{attribute addProperty BoxType "EK1100-0000-0018"}
{attribute addProperty Id "Beckhoff_ELXxxxxEK1122Beckhoff_ELXxxxxEK1122_CE175A58162A_0001_ELX1052_0000_0016ELX1052_0A1DBF07648A_0002_ELX1054_0000_0016ELX1054_FE7182BE12816A_0003_ELX1058_0000_0016ELX1058_F462A61522428A_0004_ELX2002_0000_0016ELX2002_B180A8D3405A_0005_ELX2008_0000_0016ELX2008_04E0E56B8811A_0006_ELX3152_0000_0016ELX3152_1C870F0C16020A_0007_ELX3152_0000_0017ELX3152_1C870F0C16020A_0008_ELX3152_0090_0016ELX3152_1C870F0C16020A_0009_ELX3152_0090_0017ELX3152_1C870F0C16020A_0010_ELX3158_0000_0016ELX3158_91E9C02235244A_0011_ELX3181_0000_0016ELX3181_02AD9A7917622A_0012_ELX3181_0000_0017ELX3181_02AD9A7917622A_0013_ELX3202_0000_0016ELX3202_0EB9D2E916020A_0014_ELX3202_0090_0016ELX3202_0EB9D2E916020A_0015_ELX3204_0000_0016ELX3204_5DC9EB4C22428A_0016_ELX3204_0090_0016ELX3204_5DC9EB4C22428A_0017_ELX3252_0000_0016ELX3252_F145ADB416020A_0018_ELX3312_0000_0016ELX3312_5B7A95F016020A_0019_ELX3312_0090_0016ELX3312_5B7A95F016020A_0020_ELX3314_0000_0016ELX3314_2E54E3B022428A_0021_ELX3314_0090_0016ELX3314_2E54E3B022428A_0022_ELX3351_0000_0016ELX3351_537A111616020A_0023_ELX3351_0090_0016ELX3351_537A111616020A_0024_ELX4154_0000_0016ELX4154_253CF8AE15219A_0025_ELX4181_0000_0016ELX4181_E6374D8B15219A_0026_ELX4181_0000_0017ELX4181_E6374D8B15219A_0027_ELX5151_0000_0016ELX5151_347031A716020A_0028_ELX5151_0090_0016ELX5151_347031A716020A_0030_ELX9410_0000_0016ELX9410_D787878A486A_0031_ELX9410_0000_0017ELX9410_D787878A486A_0032_ELX9410_0000_0018ELX9410_AF51CCF7486A_0033_ELX9560_0000_0016ELX9560_FB68D8D1486A_0034_ELX9560_0000_0017ELX9560_FB68D8D1486A_0035_ELX9560_0000_0018ELX9560_E7D0746E486"}
{attribute addProperty CRC "818935286"}
{attribute addProperty SizeInBites "4984"}
{attribute addProperty SizeInBytes "623"}
TYPE Beckhoff_ELXxxxx_30CFF5F6 EXTENDS EK1100_179A0949 :
STRUCT
	{attribute addProperty Name "Beckhoff_ELXxxxxEK1122"}
	Beckhoff_ELXxxxxEK1122 : Beckhoff_ELXxxxxEK1122_CE175A58;
	{attribute addProperty Name "A_0001_ELX1052_0000_0016"}
	A_0001_ELX1052_0000_0016 : ELX1052_0A1DBF07;
	{attribute addProperty Name "A_0002_ELX1054_0000_0016"}
	A_0002_ELX1054_0000_0016 : ELX1054_FE7182BE;
	{attribute addProperty Name "A_0003_ELX1058_0000_0016"}
	A_0003_ELX1058_0000_0016 : ELX1058_F462A615;
	{attribute addProperty Name "A_0004_ELX2002_0000_0016"}
	A_0004_ELX2002_0000_0016 : ELX2002_B180A8D3;
	{attribute addProperty Name "A_0005_ELX2008_0000_0016"}
	A_0005_ELX2008_0000_0016 : ELX2008_04E0E56B;
	{attribute addProperty Name "A_0006_ELX3152_0000_0016"}
	A_0006_ELX3152_0000_0016 : ELX3152_1C870F0C;
	{attribute addProperty Name "A_0007_ELX3152_0000_0017"}
	A_0007_ELX3152_0000_0017 : ELX3152_1C870F0C;
	{attribute addProperty Name "A_0008_ELX3152_0090_0016"}
	A_0008_ELX3152_0090_0016 : ELX3152_1C870F0C;
	{attribute addProperty Name "A_0009_ELX3152_0090_0017"}
	A_0009_ELX3152_0090_0017 : ELX3152_1C870F0C;
	{attribute addProperty Name "A_0010_ELX3158_0000_0016"}
	A_0010_ELX3158_0000_0016 : ELX3158_91E9C022;
	{attribute addProperty Name "A_0011_ELX3181_0000_0016"}
	A_0011_ELX3181_0000_0016 : ELX3181_02AD9A79;
	{attribute addProperty Name "A_0012_ELX3181_0000_0017"}
	A_0012_ELX3181_0000_0017 : ELX3181_02AD9A79;
	{attribute addProperty Name "A_0013_ELX3202_0000_0016"}
	A_0013_ELX3202_0000_0016 : ELX3202_0EB9D2E9;
	{attribute addProperty Name "A_0014_ELX3202_0090_0016"}
	A_0014_ELX3202_0090_0016 : ELX3202_0EB9D2E9;
	{attribute addProperty Name "A_0015_ELX3204_0000_0016"}
	A_0015_ELX3204_0000_0016 : ELX3204_5DC9EB4C;
	{attribute addProperty Name "A_0016_ELX3204_0090_0016"}
	A_0016_ELX3204_0090_0016 : ELX3204_5DC9EB4C;
	{attribute addProperty Name "A_0017_ELX3252_0000_0016"}
	A_0017_ELX3252_0000_0016 : ELX3252_F145ADB4;
	{attribute addProperty Name "A_0018_ELX3312_0000_0016"}
	A_0018_ELX3312_0000_0016 : ELX3312_5B7A95F0;
	{attribute addProperty Name "A_0019_ELX3312_0090_0016"}
	A_0019_ELX3312_0090_0016 : ELX3312_5B7A95F0;
	{attribute addProperty Name "A_0020_ELX3314_0000_0016"}
	A_0020_ELX3314_0000_0016 : ELX3314_2E54E3B0;
	{attribute addProperty Name "A_0021_ELX3314_0090_0016"}
	A_0021_ELX3314_0090_0016 : ELX3314_2E54E3B0;
	{attribute addProperty Name "A_0022_ELX3351_0000_0016"}
	A_0022_ELX3351_0000_0016 : ELX3351_537A1116;
	{attribute addProperty Name "A_0023_ELX3351_0090_0016"}
	A_0023_ELX3351_0090_0016 : ELX3351_537A1116;
	{attribute addProperty Name "A_0024_ELX4154_0000_0016"}
	A_0024_ELX4154_0000_0016 : ELX4154_253CF8AE;
	{attribute addProperty Name "A_0025_ELX4181_0000_0016"}
	A_0025_ELX4181_0000_0016 : ELX4181_E6374D8B;
	{attribute addProperty Name "A_0026_ELX4181_0000_0017"}
	A_0026_ELX4181_0000_0017 : ELX4181_E6374D8B;
	{attribute addProperty Name "A_0027_ELX5151_0000_0016"}
	A_0027_ELX5151_0000_0016 : ELX5151_347031A7;
	{attribute addProperty Name "A_0028_ELX5151_0090_0016"}
	A_0028_ELX5151_0090_0016 : ELX5151_347031A7;
	{attribute addProperty Name "A_0030_ELX9410_0000_0016"}
	A_0030_ELX9410_0000_0016 : ELX9410_D787878A;
	{attribute addProperty Name "A_0031_ELX9410_0000_0017"}
	A_0031_ELX9410_0000_0017 : ELX9410_D787878A;
	{attribute addProperty Name "A_0032_ELX9410_0000_0018"}
	A_0032_ELX9410_0000_0018 : ELX9410_AF51CCF7;
	{attribute addProperty Name "A_0033_ELX9560_0000_0016"}
	A_0033_ELX9560_0000_0016 : ELX9560_FB68D8D1;
	{attribute addProperty Name "A_0034_ELX9560_0000_0017"}
	A_0034_ELX9560_0000_0017 : ELX9560_FB68D8D1;
	{attribute addProperty Name "A_0035_ELX9560_0000_0018"}
	A_0035_ELX9560_0000_0018 : ELX9560_E7D0746E;
END_STRUCT
END_TYPE

(* stored: Version 1.2.0.0, ProductVersion 3.1.4024.9
   DUT Beckhoff_ELXxxxx_30CFF5F6: Id {5f927b3c-3393-451d-8219-f40dd7e5617b} *)
